FUNCTION_BLOCK Test_FB_Counter_Increments EXTENDS T_UnitTestBase
VAR
    Counter : CTU;
END_VAR

// Setup..
Counter(
	CU:= FALSE, 
	RESET:= TRUE, 
	PV:= , 
	Q=> , 
	CV=> );

// Test... 
Counter(
	CU:= TRUE, 
	RESET:= FALSE, 
	PV:= , 
	Q=> , 
	CV=> );
// Verify...   
Assertion.AssertEquals_WORD(
    Expected:= 1, 
    Actual:= Counter.CV, 
    VariableName:= 'Counter.CV');   

// Done...   
TestFinished();

END_FUNCTION_BLOCK

(* stored: Version 1.1.0.1, ProductVersion 3.1.4024.6
   POU Test_FB_Counter_Increments: Id {ed7d4b18-0e41-4ad1-835d-cb8be51dbc2d}, SpecialFunc None *)
